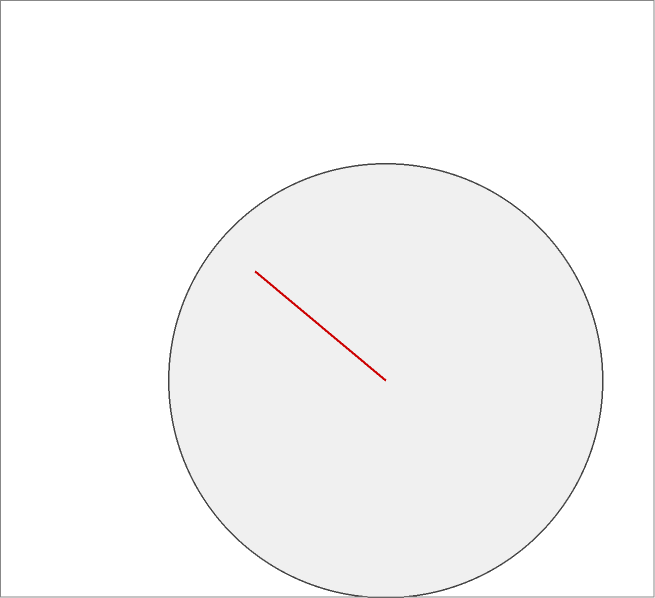
VISUALIZATION Visualization  // 655x598
    Meter180 (116,163 539x435), value: pc.MBRegs[0], style: Meter-Meter180-Gray, scale format: %.1f, scale 0..900
END_VISUALIZATION

(* stored: Version 1.1.0.1, ProductVersion 3.1.4024.12
   Visu Visualization: Id {00dfd9a0-c480-4331-9395-f872468aa2f8} *)
